// TIA Portal V16 export
// export: Created 2022-01-12T14:34:27.3129628Z, ExportSetting WithDefaults, DisplayName Totally Integrated Automation Portal, DisplayVersion V16 Update 4, DisplayName TIA Portal Version Control Interface, DisplayVersion V16 Update 2, DisplayName TIA Portal Openness, DisplayVersion V16 Update 4, DisplayName STEP 7 Professional, DisplayVersion V16 Update 4, DisplayName STEP 7 Safety, DisplayVersion V16, DisplayName WinCC Professional, DisplayVersion V16 Update 4
TYPE "typRecepturaStacjiMycia"
// stored: IsFailsafeCompliant false
   STRUCT
      nazwaReceptury : WString[33] := WSTRING#'nazwa receptury';
      Krok { S7_SetPoint := 'True'} : Array[0..6] of "typKrokRecepturyStacjiMycia";
   END_STRUCT;
   // Krok[0].nazwaKroku := WSTRING#'';
   // Krok[1].nazwaKroku := WSTRING#'Płukanie Zimne';
   // Krok[2].nazwaKroku := WSTRING#'Płukanie Gorące';
   // Krok[3].nazwaKroku := WSTRING#'Ług';
   // Krok[4].nazwaKroku := WSTRING#'Kwas';
   // Krok[5].nazwaKroku := WSTRING#'Płukanie Główne';
   // Krok[6].nazwaKroku := WSTRING#'Dezynfekcja';
END_TYPE
